// TIA Portal V20 export
TYPE "LER_FlexNet_Data"
// stored: Access Published
   STRUCT
      PUN : String[20];   // PUN
      GM_PartNumber : String[8];   // GM Part Number
      OptionalData : String[12];   // Optional Data
      TrackingID1 : String[32];   // Tracking ID1 / Component 1 of the parent
      TrackingID1Attribute : String[20];   // Tracking ID1 Attribute / Component 1 Attribute of the parent
      TrackingID2 : String[32];   // Tracking ID2 / Component 2 of the parent
      TrackingID2Attribute : String[20];   // Tracking ID2 Attribute / Component 2 Attribute of the parent
      TrackingID3 : String[32];   // Tracking ID3 / Component 3 of the parent
      TrackingID3Attribute : String[20];   // Tracking ID3 Attribute / Component 3 Attribute of the parent
      TrackingID4 : String[32];   // Tracking ID4 / Component 4 of the parent
      TrackingID4Attribute : String[20];   // Tracking ID4 Attribute / Component 4 Attribute of the parent
      TrackingID5 : String[32];   // Tracking ID5 / Component 5 of the parent
      TrackingID5Attribute : String[20];   // Tracking ID5 Attribute / Component 5 Attribute of the parent
      TrackingID6 : String[32];   // Tracking ID6 / Component 6 of the parent
      TrackingID6Attribute : String[20];   // Tracking ID6 Attribute / Component 6 Attribute of the parent
      TrackingID7 : String[32];   // Tracking ID7 / Component 7 of the parent
      TrackingID7Attribute : String[20];   // Tracking ID7 Attribute / Component 7 Attribute of the parent
      TrackingID8 : String[32];   // Tracking ID8 / Component 8 of the parent
      TrackingID8Attribute : String[20];   // Tracking ID8 Attribute / Component 8 Attribute of the parent
      TrackingID9 : String[32];   // Tracking ID9 / Component 9 of the parent
      TrackingID9Attribute : String[20];   // Tracking ID9 Attribute / Component 9 Attribute of the parent
      TrackingID10 : String[32];   // Tracking ID10 / Component 10 of the parent
      TrackingID10Attribute : String[20];   // Tracking ID10 Attribute / Component 10 Attribute of the parent
      PassFailFlagsByte : Char;   // Pass or Fail Flag Byte
      Genealogy_Cnt : Byte;   // Genealogy Count
      TransactionType : Byte;   // Transaction Type
      DataReady : Bool;   // Data Ready
      Bypassed_Fault : Bool;   // Bypassed Fault
      DataReceivedByHost : Bool;   // Data Received By Host
      ParentPartIsGood : Bool;   // Parent Part Is Good
      ParentPartOnHold : Bool;   // Parent Part On Hold
      TrackingComponent_1_IsGood : Bool;   // Tracking Component 1 Is Good
      TrackingComponent_1_OnHold : Bool;   // Tracking Component 1 On Hold
      TrackingComponent_2_IsGood : Bool;   // Tracking Component 2 Is Good
      TrackingComponent_2_OnHold : Bool;   // Tracking Component 2 On Hold
      TrackingComponent_3_IsGood : Bool;   // Tracking Component 3 Is Good
      TrackingComponent_3_OnHold : Bool;   // Tracking Component 3 On Hold
      TrackingComponent_4_IsGood : Bool;   // Tracking Component 4 Is Good
      TrackingComponent_4_OnHold : Bool;   // Tracking Component 4 On Hold
      TrackingComponent_5_IsGood : Bool;   // Tracking Component 5 Is Good
      TrackingComponent_5_OnHold : Bool;   // Tracking Component 5 On Hold
      TrackingComponent_6_IsGood : Bool;   // Tracking Component 6 Is Good
      TrackingComponent_6_OnHold : Bool;   // Tracking Component 6 On Hold
      TrackingComponent_7_IsGood : Bool;   // Tracking Component 7 Is Good
      TrackingComponent_7_OnHold : Bool;   // Tracking Component 7 On Hold
      TrackingComponent_8_IsGood : Bool;   // Tracking Component 8 Is Good
      TrackingComponent_8_OnHold : Bool;   // Tracking Component 8 On Hold
      TrackingComponent_9_IsGood : Bool;   // Tracking Component 9 Is Good
      TrackingComponent_9_OnHold : Bool;   // Tracking Component 9 On Hold
      TrackingComponent_10_IsGood : Bool;   // Tracking Component 10 Is Good
      TrackingComponent_10_OnHold : Bool;   // Tracking Component 10 On Hold
      White_LT_Solid : Bool;   // White Light Solid
      White_LT_Flash : Bool;   // White Light Flash
      Green_LT_Solid : Bool;   // Green Light Solid
      Buzzer_Output : Bool;   // Buzzer Output
      TimeStampYear : UInt;   // Time Stamp Year
      TimeStampMonth : USInt;   // Time Stamp Month
      TimeStampDate : USInt;   // Time Stamp Date
      TimeStampHour : USInt;   // Time Stamp Hour
      TimeStampMinute : USInt;   // Time Stamp Minute
      TimeStampSecond : USInt;   // Time Stamp Second
      Major_Spec_Version : Array[1..4] of Char;
      Minor_Spec_Version : Array[1..4] of Char;
      AOI_Revision : Int;   // AOI Revision
      PartPass : Bool;   // Part Pass
      PartFail : Bool;   // Part Fail
      DataReset : Bool;   // Data Reset
      DryCycle : Bool;   // Dry Cycle
      HQ_NOK : Bool;   // HQ NOK
      HQ_OK : Bool;   // HQ OK
      ReTrigger_DataReady : Bool;   // Retrigger Data Ready for Recovery
   END_STRUCT;
END_TYPE
